{attribute 'qualified_only'}
VAR_GLOBAL CONSTANT
	cMaxInv : UINT:=12; //Maksymalna liczba inverterow
END_VAR

(* stored: Version 1.1.0.1, ProductVersion 3.1.4024.16
   GVL GVL_Inverter: Id {79b6121c-8beb-4d5d-b8c2-5d43410ef7da} *)
